FUNCTION_BLOCK FB_ReplaceLongStringCharTests EXTENDS FB_TestSuite

//==============================================================
//MAIN TESTS
//==============================================================

testMain01_ExtractCharFromLongString_AllCahrsExtracted();
testMain02_RepalceCharFromLongString_AllCahrsRepalced();

//==============================================================
//NEGATIVE TESTS
//==============================================================

testNeg01_ReplaceInputs_NoChangeInFullCode();
testNeg02_TwoCharsOnInputs_OneCharReplaced();

//==============================================================
//SEQUENCE TESTS
//==============================================================

//==============================================================
//OTHERS TESTS
//==============================================================

METHOD INTERNAL testMain01_ExtractCharFromLongString_AllCahrsExtracted
VAR
	
	sFullCode			: T_LongSTRING;	
	sExpectedResult		: T_LongSTRING;
	sActualResult		: T_LongSTRING;
END_VAR
TEST('testMain01_ExtractCharFromLongString_AllCahrsExtracted');

sFullCode := 'ST=53;$02CT=10;DS=GZDNP5JOA3IL$1D;OG=3;XP=-50;YP=50;AP=-88;CS=06.2;SC=0070;QS=3;PN=1;$03$04
											ST=53;$02CT=10;DS=N7E1Y89UNK3O$1D;OG=3;XP=-50;YP=-50;AP=-88;CS=06.2;SC=0070;QS=3;PN=2;$03$04
											ST=53;$02CT=10;DS=JHWJXYFNX9DS$1D;OG=3;XP=50;YP=50;AP=-88;CS=06.2;SC=0070;QS=3;PN=3;$03$04
											ST=53;$02CT=10;DS=XGBEZLBV8A9I$1D;OG=3;XP=50;YP=-50;AP=-88;CS=06.2;SC=0070;QS=3;PN=4;$03$04'; 

sExpectedResult := 'ST=53;$02CT=10;DS=GZDNP5JOA3IL;OG=3;XP=-50;YP=50;AP=-88;CS=06.2;SC=0070;QS=3;PN=1;$03$04
											ST=53;$02CT=10;DS=N7E1Y89UNK3O;OG=3;XP=-50;YP=-50;AP=-88;CS=06.2;SC=0070;QS=3;PN=2;$03$04
											ST=53;$02CT=10;DS=JHWJXYFNX9DS;OG=3;XP=50;YP=50;AP=-88;CS=06.2;SC=0070;QS=3;PN=3;$03$04
											ST=53;$02CT=10;DS=XGBEZLBV8A9I;OG=3;XP=50;YP=-50;AP=-88;CS=06.2;SC=0070;QS=3;PN=4;$03$04'; 


sActualResult	:= F_ReplaceLongSingleChar(sFullCode:= sFullCode, 
							sCharRemove:= '$1D', 
							sReplacmentChar:='' );
							
AssertEquals_STRING(Expected:= sExpectedResult, 
						Actual:= sActualResult, 
						Message:= 'Extracted string is not as expected');
						
TEST_FINISHED();
END_METHOD

METHOD INTERNAL testMain02_RepalceCharFromLongString_AllCahrsRepalced
VAR
	
	sFullCode			: T_LongSTRING;	
	sExpectedResult		: T_LongSTRING;
	sActualResult		: T_LongSTRING;
END_VAR
TEST('testMain02_RepalceCharFromLongString_AllCahrsRepalced');

sFullCode := 'ST=53;$02CT=10;DS=GZDNP5JOA3IL$1D;OG=3;XP=-50;YP=50;AP=-88;CS=06.2;SC=0070;QS=3;PN=1;$03$04
											ST=53;$02CT=10;DS=N7E1Y89UNK3O$1D;OG=3;XP=-50;YP=-50;AP=-88;CS=06.2;SC=0070;QS=3;PN=2;$03$04
											ST=53;$02CT=10;DS=JHWJXYFNX9DS$1D;OG=3;XP=50;YP=50;AP=-88;CS=06.2;SC=0070;QS=3;PN=3;$03$04
											ST=53;$02CT=10;DS=XGBEZLBV8A9I$1D;OG=3;XP=50;YP=-50;AP=-88;CS=06.2;SC=0070;QS=3;PN=4;$03$04'; 

sExpectedResult := 'ST=53;$02CT=10;DS=GZDNP5JAA3IL$1D;AG=3;XP=-50;YP=50;AP=-88;CS=06.2;SC=0070;QS=3;PN=1;$03$04
											ST=53;$02CT=10;DS=N7E1Y89UNK3A$1D;AG=3;XP=-50;YP=-50;AP=-88;CS=06.2;SC=0070;QS=3;PN=2;$03$04
											ST=53;$02CT=10;DS=JHWJXYFNX9DS$1D;AG=3;XP=50;YP=50;AP=-88;CS=06.2;SC=0070;QS=3;PN=3;$03$04
											ST=53;$02CT=10;DS=XGBEZLBV8A9I$1D;AG=3;XP=50;YP=-50;AP=-88;CS=06.2;SC=0070;QS=3;PN=4;$03$04'; 


sActualResult	:= F_ReplaceLongSingleChar(sFullCode:= sFullCode, 
							sCharRemove:= 'O', 
							sReplacmentChar:='A' );
							
AssertEquals_STRING(Expected:= sExpectedResult, 
						Actual:= sActualResult, 
						Message:= 'Extracted string is not as expected');
						
TEST_FINISHED();
END_METHOD

METHOD INTERNAL testNeg01_ReplaceInputs_NoChangeInFullCode
VAR
	
	sFullCode			: T_LongSTRING;	
	sExpectedResult		: T_LongSTRING;
	sActualResult		: T_LongSTRING;
END_VAR
TEST('testNeg01_ReplaceInputs_NoChangeInFullCode');

sFullCode := 'ST=53;$02CT=10;DS=GZDNP5JOA3IL$1D;OG=3;XP=-50;YP=50;AP=-88;CS=06.2;SC=0070;QS=3;PN=1;$03$04
											ST=53;$02CT=10;DS=N7E1Y89UNK3O$1D;OG=3;XP=-50;YP=-50;AP=-88;CS=06.2;SC=0070;QS=3;PN=2;$03$04
											ST=53;$02CT=10;DS=JHWJXYFNX9DS$1D;OG=3;XP=50;YP=50;AP=-88;CS=06.2;SC=0070;QS=3;PN=3;$03$04
											ST=53;$02CT=10;DS=XGBEZLBV8A9I$1D;OG=3;XP=50;YP=-50;AP=-88;CS=06.2;SC=0070;QS=3;PN=4;$03$04'; 

sExpectedResult := 'ST=53;$02CT=10;DS=GZDNP5JOA3IL$1D;OG=3;XP=-50;YP=50;AP=-88;CS=06.2;SC=0070;QS=3;PN=1;$03$04
											ST=53;$02CT=10;DS=N7E1Y89UNK3O$1D;OG=3;XP=-50;YP=-50;AP=-88;CS=06.2;SC=0070;QS=3;PN=2;$03$04
											ST=53;$02CT=10;DS=JHWJXYFNX9DS$1D;OG=3;XP=50;YP=50;AP=-88;CS=06.2;SC=0070;QS=3;PN=3;$03$04
											ST=53;$02CT=10;DS=XGBEZLBV8A9I$1D;OG=3;XP=50;YP=-50;AP=-88;CS=06.2;SC=0070;QS=3;PN=4;$03$04'; 


sActualResult	:= F_ReplaceLongSingleChar(sFullCode:= sFullCode, 
							sCharRemove:= '', 
							sReplacmentChar:='$1D' );
							
AssertEquals_STRING(Expected:= sExpectedResult, 
						Actual:= sActualResult, 
						Message:= 'Extracted string is not as expected');
						
TEST_FINISHED();
END_METHOD

METHOD INTERNAL testNeg02_TwoCharsOnInputs_OneCharReplaced
VAR
	
	sFullCode			: T_LongSTRING;	
	sExpectedResult		: T_LongSTRING;
	sActualResult		: T_LongSTRING;
END_VAR
TEST('testNeg02_TwoCharsOnInputs_OneCharReplaced');

sFullCode := 'ST=53;$02CT=10;DS=GZDNP5JOA3IL$1D;OG=3;XP=-50;YP=50;AP=-88;CS=06.2;SC=0070;QS=3;PN=1;$03$04
											ST=53;$02CT=10;DS=N7E1Y89UNK3O$1D;OG=3;XP=-50;YP=-50;AP=-88;CS=06.2;SC=0070;QS=3;PN=2;$03$04
											ST=53;$02CT=10;DS=JHWJXYFNX9DS$1D;OG=3;XP=50;YP=50;AP=-88;CS=06.2;SC=0070;QS=3;PN=3;$03$04
											ST=53;$02CT=10;DS=XGBEZLBV8A9I$1D;OG=3;XP=50;YP=-50;AP=-88;CS=06.2;SC=0070;QS=3;PN=4;$03$04'; 

sExpectedResult := 'ST=53;$02CT=10;DS=GZDNP5JOA3IL$1D;OG=3;XP=-50;YP=50;AP=-88;CS=06.2;SC=0070;QS=3;PN=1;$1D$04
											ST=53;$02CT=10;DS=N7E1Y89UNK3O$1D;OG=3;XP=-50;YP=-50;AP=-88;CS=06.2;SC=0070;QS=3;PN=2;$1D$04
											ST=53;$02CT=10;DS=JHWJXYFNX9DS$1D;OG=3;XP=50;YP=50;AP=-88;CS=06.2;SC=0070;QS=3;PN=3;$1D$04
											ST=53;$02CT=10;DS=XGBEZLBV8A9I$1D;OG=3;XP=50;YP=-50;AP=-88;CS=06.2;SC=0070;QS=3;PN=4;$1D$04';


{warning disable C0198}

sActualResult	:= F_ReplaceLongSingleChar(sFullCode:= sFullCode, 
							sCharRemove:= '$03$04', 
							sReplacmentChar:='$1D' );
{warning restore C0198}	
						
AssertEquals_STRING(Expected:= sExpectedResult, 
						Actual:= sActualResult, 
						Message:= 'Extracted string is not as expected');
						
TEST_FINISHED();
END_METHOD

END_FUNCTION_BLOCK

(* stored: Version 1.1.0.1
   POU FB_ReplaceLongStringCharTests: Id {25c5792a-3d1a-4c1f-a871-0deacf66dcbc}, SpecialFunc None
   Folder 01 Main: Id {e30b7842-edff-4093-a303-9ff2f550a3a7}
   Folder 02 Negative: Id {94fd32b4-85ac-42ca-946e-a66ebb289ccd}
   Method testMain01_ExtractCharFromLongString_AllCahrsExtracted: Id {70a70862-120d-408d-9d00-93959ac3bab5}
   Method testMain02_RepalceCharFromLongString_AllCahrsRepalced: Id {5406bdd6-18a3-42dc-b037-eb6fc9c388a1}
   Method testNeg01_ReplaceInputs_NoChangeInFullCode: Id {8c5bfa65-17a3-470a-a0f3-4d0cbd4263f6}
   Method testNeg02_TwoCharsOnInputs_OneCharReplaced: Id {b2e4f6ad-8fee-4e58-9ae8-5b4fc405f3ab} *)
